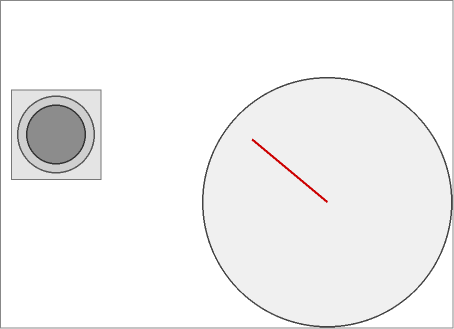
VISUALIZATION Visualization  // 454x329
    PushSwitchLed (11,64 90x141), variable: .MAIN.MxOn, behaviour: TOGGLE, style: Switch-PushSwitchLed-Gray
    Meter180 (202,77 250x250), style: Meter-Meter180-Gray, scale format: %.1f, scale 0..1000
END_VISUALIZATION

(* stored: Version 1.1.0.1, ProductVersion 3.1.4020.6
   Visu Visualization: Id {c7f871f7-1935-48d9-bcb4-fcb1bb905786} *)
